Fanuc KAREL source: kb00035.KL

-- PROVISIONAL review KL for V770-1; original PC SHA256 a2e807b825838350bbb4f590480c6562b1a82986250faed03aa167a501377d2a
-- Incomplete behavior may be omitted. Consult companion uncertainty JSON. Do not deploy.
PROGRAM KB00035
%NOLOCKGROUP
BEGIN
  -- UNRESOLVED_PC offsets 5-12; opcodes 9D,23
  -- UNRESOLVED_PC offsets 17-24; opcodes 9D,23
  -- UNRESOLVED_PC offsets 29-36; opcodes 9D,23
  -- UNRESOLVED_PC offsets 41-50; opcodes 3F,75
  -- UNRESOLVED_PC offsets 55-85; opcodes 27,22,22,22,22,2A,31
  -- UNRESOLVED_PC offsets 90-94; opcodes 7F
END KB00035
